TYPE EM :
STRUCT
	
	MesEActCons				: REAL ; 		(* Value of Active Energy consumed		*)
	MesEActProd				: REAL ;		(* Value of Active Energy produced      *)
	MesEReactCons			: REAL ;		(* Value of Reactive Energy consumed    *)
	MesEReactProd			: REAL ;		(* Value of Reactive Energy produced    *)
	                                                                             
	MesAlarmCode			: WORD ;	 	(* (NA) Internal Akuo AlarmCode         *)
	MesWarningCode			: WORD ; 		(* (NA) Internal Akuo WarningCode       *)
	MesEventCode			: WORD ; 		(* (NA) Internal Akuo EventCode	        *)

END_STRUCT
END_TYPE

(* stored: Version 1.1.0.1, ProductVersion 3.1.4024.6
   DUT EM: Id {55b9897b-27a6-4b7b-956d-678b5171c54d} *)
